// TIA Portal V16 export
// export: Created 2022-11-17T11:55:35.8376525Z, ExportSetting WithDefaults, DisplayName Totally Integrated Automation Portal, DisplayVersion V16 Update 6, DisplayName TIA Portal Version Control Interface, DisplayVersion V16 Update 2, DisplayName TIA Portal Openness, DisplayVersion V16 Update 6, DisplayName SINAMICS Startdrive Advanced, DisplayVersion V16 Update 5, DisplayName SINAMICS Startdrive G130, G150, S120, S150, SINAMICS MV, S210, DisplayVersion V16 Update 5, DisplayName SINAMICS Startdrive G110M, G120, G120C, G120D, G120P, G115D, DisplayVersion V16 Update 5, DisplayName STEP 7 Professional, DisplayVersion V16 Update 6, DisplayName STEP 7 Safety, DisplayVersion V16, DisplayName WinCC Advanced, DisplayVersion V16 Update 6
DATA_BLOCK "DB251_ProgramDisplay"   // DB251
{ S7_Optimized_Access := 'FALSE' }
VERSION : 0.0
// stored: AutoNumber false, IsOnlyStoredInLoadMemory false, IsWriteProtectedInAS false
   VAR RETAIN
      Display { S7_SetPoint := 'True'} : "DatiProgramma";
   END_VAR
BEGIN
   Display.Wrapping := TRUE;
   Display.TopLenght := 500;
   Display.TopRelease := 0;
   Display.TopDown := 0;
   Display.Top := 4;
   Display.PressurePTime := 0;
   Display.LifterTime := 0;
   Display.RevOverContrast := 1;
   Display.RopeEndCycle := 16#02;
   Display.Spare4 := 16#01;
   Display.RopeTime := 1500;
   Display.RevOverClamp := 1;
   Display.FilmForceFinalRev := 10;
   Display.FilmPrestretchFinalRev := 100;
   Display.ArmSpeed := 100;
   Display.CarriageDown4Top := 500;
   Display.TopDownTime := 1500;
   Display.LapsUnderTop := 0;
   Display.Spare6 := 0;
   Display.Spare7 := 0;
   Display.Spare8 := 0;
   Display.Spare9 := 0;
   Display.Spare10 := 0;
   Display.Spare11 := 0;
   Display.Spare12 := 0;
   Display.Overlap0_1 := 0;
   Display.Height1 := 130;
   Display.Landmark1 := FALSE;
   Display.Lifter1 := FALSE;
   Display.SpareBit1H1 := FALSE;
   Display.Airblower1 := TRUE;
   Display.NextStep1 := TRUE;
   Display.PressureP1 := TRUE;
   Display.SpareByte2H1 := 16#00;
   Display.Revolution1 := 1;
   Display.RopeUnit1_1 := 16#01;
   Display.RopeUnit1_2 := 16#01;
   Display.FilmForce1 := 5;
   Display.FilmPrestretch1 := 200;
   Display.Spare3H1 := 0;
   Display.Spare49 := 0;
   Display.Spare50 := 0;
   Display.Spare51 := 0;
   Display.Spare52 := 0;
   Display.Spare53 := 0;
   Display.Overlap1_2 := 0;
   Display.Height2 := 50;
   Display.Landmark2 := FALSE;
   Display.Lifter2 := FALSE;
   Display.SpareBit1H2 := FALSE;
   Display.Airblower2 := TRUE;
   Display.NextStep2 := TRUE;
   Display.PressureP2 := TRUE;
   Display.SpareByte2H2 := 16#00;
   Display.Revolution2 := 1;
   Display.RopeUnit2_1 := 16#01;
   Display.RopeUnit2_2 := 16#01;
   Display.FilmForce2 := 20;
   Display.FilmPrestretch2 := 200;
   Display.Spare3H2 := 0;
   Display.Spare54 := 0;
   Display.Spare55 := 0;
   Display.Spare56 := 0;
   Display.Spare57 := 0;
   Display.Spare58 := 0;
   Display.Overlap2_3 := 100;
   Display.Height3 := -50;
   Display.Landmark3 := TRUE;
   Display.Lifter3 := FALSE;
   Display.SpareBit1H3 := FALSE;
   Display.Airblower3 := TRUE;
   Display.NextStep3 := TRUE;
   Display.PressureP3 := TRUE;
   Display.SpareByte2H3 := 16#00;
   Display.Revolution3 := 2;
   Display.RopeUnit3_1 := 16#01;
   Display.RopeUnit3_2 := 16#01;
   Display.FilmForce3 := 30;
   Display.FilmPrestretch3 := 200;
   Display.Spare3H3 := 0;
   Display.Spare59 := 0;
   Display.Spare60 := 0;
   Display.Spare61 := 380;
   Display.Spare62 := 2800;
   Display.Spare63 := 0;
   Display.Overlap3_4 := 100;
   Display.Height4 := 100;
   Display.Landmark4 := FALSE;
   Display.Lifter4 := FALSE;
   Display.SpareBit1H4 := FALSE;
   Display.Airblower4 := TRUE;
   Display.NextStep4 := TRUE;
   Display.PressureP4 := TRUE;
   Display.SpareByte2H4 := 16#00;
   Display.Revolution4 := 3;
   Display.RopeUnit4_1 := 16#02;
   Display.RopeUnit4_2 := 16#02;
   Display.FilmForce4 := 30;
   Display.FilmPrestretch4 := 200;
   Display.Spare3H4 := 0;
   Display.Spare64 := 0;
   Display.Spare65 := 0;
   Display.Spare66 := 0;
   Display.Spare67 := 0;
   Display.Spare68 := 0;
   Display.Overlap4_5 := 0;
   Display.Height5 := 50;
   Display.Landmark5 := FALSE;
   Display.Lifter5 := FALSE;
   Display.SpareBit1H5 := FALSE;
   Display.Airblower5 := TRUE;
   Display.NextStep5 := FALSE;
   Display.PressureP5 := FALSE;
   Display.SpareByte2H5 := 16#00;
   Display.Revolution5 := 1;
   Display.RopeUnit5_1 := 16#01;
   Display.RopeUnit5_2 := 16#01;
   Display.FilmForce5 := 30;
   Display.FilmPrestretch5 := 200;
   Display.Spare3H5 := 0;
   Display.Spare69 := 0;
   Display.Spare70 := 0;
   Display.Spare71 := 0;
   Display.Spare72 := 0;
   Display.Spare73 := 0;
   Display.Overlap5_6 := 100;
   Display.Height6 := 50;
   Display.Landmark6 := FALSE;
   Display.Lifter6 := FALSE;
   Display.SpareBit1H6 := FALSE;
   Display.Airblower6 := TRUE;
   Display.NextStep6 := FALSE;
   Display.PressureP6 := FALSE;
   Display.SpareByte2H6 := 16#00;
   Display.Revolution6 := 2;
   Display.RopeUnit6_1 := 16#02;
   Display.RopeUnit6_2 := 16#01;
   Display.FilmForce6 := 20;
   Display.FilmPrestretch6 := 200;
   Display.Spare3H6 := 0;
   Display.Spare74 := 0;
   Display.Spare75 := 0;
   Display.Spare76 := 0;
   Display.Spare77 := 0;
   Display.Spare78 := 0;
   Display.Overlap6_7 := 0;
   Display.Height7 := 0;
   Display.Landmark7 := FALSE;
   Display.Lifter7 := FALSE;
   Display.SpareBit1H7 := FALSE;
   Display.Airblower7 := FALSE;
   Display.NextStep7 := TRUE;
   Display.PressureP7 := FALSE;
   Display.SpareByte2H7 := 16#00;
   Display.Revolution7 := 1;
   Display.RopeUnit7_1 := 16#01;
   Display.RopeUnit7_2 := 16#01;
   Display.FilmForce7 := 0;
   Display.FilmPrestretch7 := 100;
   Display.Spare3H7 := 0;
   Display.Spare79 := 0;
   Display.Spare80 := 0;
   Display.Spare81 := 0;
   Display.Spare82 := 0;
   Display.Spare83 := 0;
   Display.Overlap7_8 := 0;
   Display.Height8 := 0;
   Display.Landmark8 := FALSE;
   Display.Lifter8 := FALSE;
   Display.SpareBit1H8 := FALSE;
   Display.Airblower8 := FALSE;
   Display.NextStep8 := TRUE;
   Display.PressureP8 := FALSE;
   Display.SpareByte2H8 := 16#00;
   Display.Revolution8 := 1;
   Display.RopeUnit8_1 := 16#01;
   Display.RopeUnit8_2 := 16#01;
   Display.FilmForce8 := 0;
   Display.FilmPrestretch8 := 100;
   Display.Spare3H8 := 0;
   Display.Spare84 := 0;
   Display.Spare85 := 0;
   Display.Spare86 := 0;
   Display.Spare87 := 0;
   Display.Spare88 := 0;
   Display.Overlap8_9 := 0;
   Display.Height9 := 0;
   Display.Landmark9 := FALSE;
   Display.Lifter9 := FALSE;
   Display.SpareBit1H9 := FALSE;
   Display.Airblower9 := FALSE;
   Display.NextStep9 := TRUE;
   Display.PressureP9 := FALSE;
   Display.SpareByte2H9 := 16#00;
   Display.Revolution9 := 1;
   Display.RopeUnit9_1 := 16#01;
   Display.RopeUnit9_2 := 16#01;
   Display.FilmForce9 := 0;
   Display.FilmPrestretch9 := 100;
   Display.Spare3H9 := 0;
   Display.Spare89 := 0;
   Display.Spare90 := 0;
   Display.Spare91 := 0;
   Display.Spare92 := 0;
   Display.Spare93 := 0;
   Display.Overlap9_10 := 0;
   Display.Height10 := 0;
   Display.Landmark10 := FALSE;
   Display.Lifter10 := FALSE;
   Display.SpareBit1H10 := FALSE;
   Display.Airblower10 := FALSE;
   Display.NextStep10 := FALSE;
   Display.PressureP10 := FALSE;
   Display.SpareByte2H10 := 16#00;
   Display.Revolution10 := 1;
   Display.RopeUnit10_1 := 16#01;
   Display.RopeUnit10_2 := 16#01;
   Display.FilmForce10 := 0;
   Display.FilmPrestretch10 := 100;
   Display.Spare3H10 := 0;
   Display.Spare94 := 0;
   Display.Spare95 := 0;
   Display.Spare96 := 0;
   Display.Spare97 := 0;
   Display.Spare98 := 0;
   Display.Overlap10_11 := 0;
   Display.Height11 := 0;
   Display.Landmark11 := FALSE;
   Display.Lifter11 := FALSE;
   Display.SpareBit1H11 := FALSE;
   Display.Airblower11 := FALSE;
   Display.NextStep11 := TRUE;
   Display.PressureP11 := FALSE;
   Display.SpareByte2H11 := 16#00;
   Display.Revolution11 := 1;
   Display.RopeUnit11_1 := 16#01;
   Display.RopeUnit11_2 := 16#01;
   Display.FilmForce11 := 0;
   Display.FilmPrestretch11 := 100;
   Display.Spare3H11 := 0;
   Display.Spare99 := 0;
   Display.Spare100 := 0;
   Display.Spare101 := 0;
   Display.Spare102 := 0;
   Display.Spare103 := 0;
   Display.Overlap11_12 := 0;
   Display.Height12 := 0;
   Display.Landmark12 := FALSE;
   Display.Lifter12 := FALSE;
   Display.SpareBit1H12 := FALSE;
   Display.Airblower12 := FALSE;
   Display.NextStep12 := FALSE;
   Display.PressureP12 := FALSE;
   Display.SpareByte2H12 := 16#00;
   Display.Revolution12 := 1;
   Display.RopeUnit12_1 := 16#01;
   Display.RopeUnit12_2 := 16#01;
   Display.FilmForce12 := 0;
   Display.FilmPrestretch12 := 100;
   Display.Spare3H12 := 0;
   Display.Spare104 := 0;
   Display.Spare105 := 0;
   Display.Spare106 := 0;
   Display.Spare107 := 0;
   Display.Spare108 := 0;
END_DATA_BLOCK
